{attribute 'linkalways'} 
{attribute 'no_explicit_call' := 'This FB is a CLASS and must be accessed using methods or properties'}
{attribute 'enable_dynamic_creation'}
FUNCTION_BLOCK FINAL GT_INT EXTENDS Node
VAR
	in1 : _INT(0);
	in2 : _INT(0);
	out : _BOOL(FALSE);
END_VAR

METHOD PUBLIC Clone : I_Node
VAR
	pNode : POINTER TO GT_INT;
END_VAR
pNode := __NEW(GT_INT);
Clone := pNode^;
END_METHOD

METHOD FB_init : BOOL
VAR_INPUT
	bInitRetains : BOOL; // if TRUE, the retain variables are initialized (warm start / cold start)
	bInCopyCode : BOOL;  // if TRUE, the instance afterwards gets moved into the copy code (online change)
END_VAR
AddInput('in1',THIS^.in1);
AddInput('in2',THIS^.in2);
AddOutput('out', THIS^.out);
END_METHOD

METHOD PROTECTED OnExecute
VAR
END_VAR
out.Value := in1.Value > in2.Value;
END_METHOD

END_FUNCTION_BLOCK

(* stored: Version 1.1.0.1, ProductVersion 3.1.4024.15
   POU GT_INT: Id {a08a7550-05bc-4ba4-b7e4-e0e1e2c73d4f}, SpecialFunc None
   Folder Constructor: Id {9bb1d753-b347-458e-bbb2-4b9c118bf48a}
   Method Clone: Id {fb05e37f-7c61-4802-86f0-b7d1b0d60c8b}
   Method FB_init: Id {4932193b-4f43-448c-ae6f-97c097bcdfef}
   Method OnExecute: Id {acfd8543-f4bc-41c8-9a43-429021f8fc9e} *)
